PROGRAM PRG_AtEntry01
VAR
	intnFBSensor : FB_Sensors;
	FEdge : F_TRIG;
	REdge : R_TRIG;
	RTrigPulse : bool;
END_VAR

intnFBSensor (
	iSensor := At_Entry_1,
	iTimeToActuateSensor := 0,
);

FEdge (
	CLK := intnFBSensor.outSensorON,
);

REdge (
	CLK :=  intnFBSensor.outSensorON,
	Q => RTrigPulse,
);

END_PROGRAM

(* stored: Version 1.1.0.1
   POU PRG_AtEntry01: Id {f61ac04f-f01d-4680-a283-4ab8a301dbdf}, SpecialFunc None *)
